// TIA Portal project "Giữa kì" (V15)

(* hardware
DEVICE "S7-1200 station_1"  S7-1200 Station
   slot 0: "Rack_0"  S7-1200 Rack  Rack  V1.0
   slot 1: "PLC_1"  CPU 1214C DC/DC/DC  6ES7 214-1AG40-0XB0  V4.2
*)

// ===== PLC "PLC_1"  CPU 1214C DC/DC/DC =====

VAR_GLOBAL   // PLC tag table "Default tag table"
   "enableSystem" AT %M0.0 : Bool;
   "iStart" AT %M0.1 : Bool;
   "iStop" AT %M0.2 : Bool;
   "oPump1" AT %Q0.0 : Bool;
   "oPump2" AT %Q0.1 : Bool;
   "mRespond" AT %M0.3 : Bool;
   "iSensorHigh1" AT %M0.4 : Bool;
   "iSensorLow1" AT %M0.5 : Bool;
   "Tag_1" AT %M100.0 : Bool;
   "Tag_2" AT %M100.1 : Bool;
   "mTank1" AT %M0.6 : Bool;
   "oPump3" AT %Q0.2 : Bool;
   "oValve1" AT %Q0.4 : Bool;
   "iSensorHigh3" AT %M1.1 : Bool;
   "iSensorLow3" AT %M1.2 : Bool;
   "iSensorHigh2" AT %M1.3 : Bool;
   "iSensorLow2" AT %M1.4 : Bool;
   "iSensorHigh4" AT %M1.5 : Bool;
   "iSensorLow4" AT %M1.6 : Bool;
   "mTank2" AT %M1.7 : Bool;
   "Tag_3" AT %M100.2 : Bool;
   "Tag_4" AT %M100.3 : Bool;
   "Tag_5" AT %M100.4 : Bool;
   "Tag_6" AT %M100.5 : Bool;
   "mTank3" AT %M2.0 : Bool;
   "mTank4" AT %M2.1 : Bool;
   "oValve2" AT %Q0.5 : Bool;
   "Tag_7" AT %M100.6 : Bool;
   "oPump4" AT %Q0.3 : Bool;
   "Tag_8" AT %M100.7 : Bool;
END_VAR

DATA_BLOCK "Data_block_1"   // DB3
{ S7_Optimized_Access := 'TRUE' }
VERSION : 0.1
   VAR
      RequiredSalinity : Real := 3.0;
      ActualSalinity : Real := 4.0;
   END_VAR
BEGIN
END_DATA_BLOCK

// folder: System blocks/Program resources

DATA_BLOCK "TimerPump1"   // DB1
{ S7_Optimized_Access := 'TRUE' }
AUTHOR : Simatic
FAMILY : IEC
NAME : IEC_TMR
VERSION : 1.0
// stored: InstanceOfName IEC_TIMER
"IEC_TIMER"
BEGIN
END_DATA_BLOCK

DATA_BLOCK "TimerPump2"   // DB2
{ S7_Optimized_Access := 'TRUE' }
AUTHOR : Simatic
FAMILY : IEC
NAME : IEC_TMR
VERSION : 1.0
// stored: InstanceOfName IEC_TIMER
"IEC_TIMER"
BEGIN
END_DATA_BLOCK

// folder: (top level)

ORGANIZATION_BLOCK "Main"   // OB1, LAD, ProgramCycle
TITLE = "Main Program Sweep (Cycle)"
{ S7_Optimized_Access := 'TRUE' }
VERSION : 0.1
   VAR_INPUT
      Initial_Call : Bool;   // Initial call of this OB
      Remanence : Bool;   // =True, if remanent data are available
   END_VAR
   VAR_TEMP   // added for the SCL form of the ladder/FBD networks
      _w1 : Bool;
      _w2 : Bool;
   END_VAR
BEGIN

REGION Network 1
   // Mở và tắt hệ thống
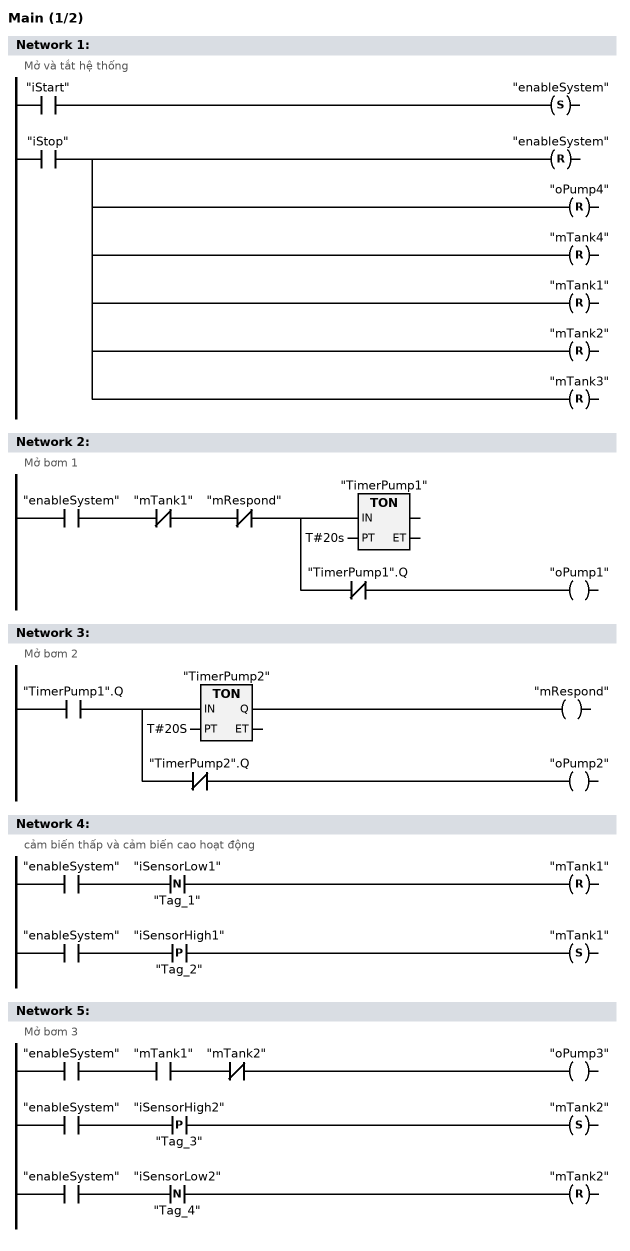
   RUNG wire#powerrail
      Contact( "iStart" )
      S_Coil( "enableSystem" )
   END_RUNG
   RUNG wire#powerrail
      Contact( "iStop" )
      wire#w1
      R_Coil( "enableSystem" )
   END_RUNG
   RUNG wire#w1
      R_Coil( "oPump4" )
   END_RUNG
   RUNG wire#w1
      R_Coil( "mTank4" )
   END_RUNG
   RUNG wire#w1
      R_Coil( "mTank1" )
   END_RUNG
   RUNG wire#w1
      R_Coil( "mTank2" )
   END_RUNG
   RUNG wire#w1
      R_Coil( "mTank3" )
   END_RUNG
   // the same network as SCL:
   IF "iStart" THEN "enableSystem" := TRUE; END_IF;
   IF "iStop" THEN
       "enableSystem" := FALSE;
       "oPump4" := FALSE;
       "mTank4" := FALSE;
       "mTank1" := FALSE;
       "mTank2" := FALSE;
       "mTank3" := FALSE;
   END_IF;
END_REGION

REGION Network 2
   // Mở bơm 1
   #_w1 := "enableSystem" AND NOT "mTank1" AND NOT "mRespond";
   "TimerPump1".TON(IN := #_w1, PT := T#20s);
   "oPump1" := #_w1 AND NOT "TimerPump1".Q;
END_REGION

REGION Network 3
   // Mở bơm 2
   "TimerPump2".TON(IN := "TimerPump1".Q, PT := T#20S);
   "mRespond" := "TimerPump2".Q;
   "oPump2" := "TimerPump1".Q AND NOT "TimerPump2".Q;
END_REGION

REGION Network 4
   // cảm biến thấp và cảm biến cao hoạt động
   RUNG wire#powerrail
      Contact( "enableSystem" )
      N_Contact(operand := "iSensorLow1", bit := "Tag_1")
      R_Coil( "mTank1" )
   END_RUNG
   RUNG wire#powerrail
      Contact( "enableSystem" )
      P_Contact(operand := "iSensorHigh1", bit := "Tag_2")
      S_Coil( "mTank1" )
   END_RUNG
   // the same network as SCL:
   #_w1 := "enableSystem" AND NOT "iSensorLow1" AND "Tag_1";   // falling edge of "iSensorLow1"
   "Tag_1" := "iSensorLow1";
   IF #_w1 THEN "mTank1" := FALSE; END_IF;
   #_w2 := "enableSystem" AND "iSensorHigh1" AND NOT "Tag_2";   // rising edge of "iSensorHigh1"
   "Tag_2" := "iSensorHigh1";
   IF #_w2 THEN "mTank1" := TRUE; END_IF;
END_REGION

REGION Network 5
   // Mở bơm 3
   RUNG wire#powerrail
      Contact( "enableSystem" )
      Contact( "mTank1" )
      I_Contact( "mTank2" )
      Coil( "oPump3" )
   END_RUNG
   RUNG wire#powerrail
      Contact( "enableSystem" )
      P_Contact(operand := "iSensorHigh2", bit := "Tag_3")
      S_Coil( "mTank2" )
   END_RUNG
   RUNG wire#powerrail
      Contact( "enableSystem" )
      N_Contact(operand := "iSensorLow2", bit := "Tag_4")
      R_Coil( "mTank2" )
   END_RUNG
   // the same network as SCL:
   "oPump3" := "enableSystem" AND "mTank1" AND NOT "mTank2";
   #_w1 := "enableSystem" AND "iSensorHigh2" AND NOT "Tag_3";   // rising edge of "iSensorHigh2"
   "Tag_3" := "iSensorHigh2";
   IF #_w1 THEN "mTank2" := TRUE; END_IF;
   #_w2 := "enableSystem" AND NOT "iSensorLow2" AND "Tag_4";   // falling edge of "iSensorLow2"
   "Tag_4" := "iSensorLow2";
   IF #_w2 THEN "mTank2" := FALSE; END_IF;
END_REGION

REGION Network 6
   // Mở van 1 cho nước xuống bể 3
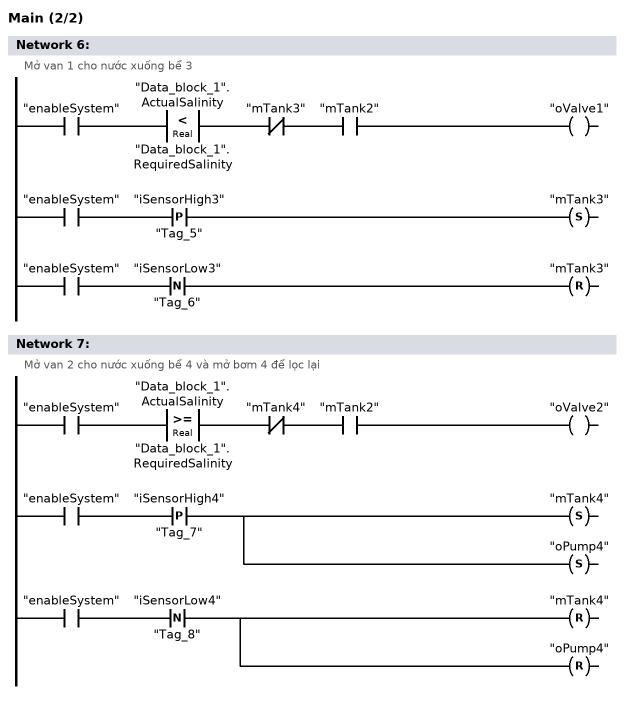
   RUNG wire#powerrail
      Contact( "enableSystem" )
      { S7_Templates := "SrcType := Real" } LT_Contact(in1 := "Data_block_1".ActualSalinity, in2 := "Data_block_1".RequiredSalinity)
      I_Contact( "mTank3" )
      Contact( "mTank2" )
      Coil( "oValve1" )
   END_RUNG
   RUNG wire#powerrail
      Contact( "enableSystem" )
      P_Contact(operand := "iSensorHigh3", bit := "Tag_5")
      S_Coil( "mTank3" )
   END_RUNG
   RUNG wire#powerrail
      Contact( "enableSystem" )
      N_Contact(operand := "iSensorLow3", bit := "Tag_6")
      R_Coil( "mTank3" )
   END_RUNG
   // the same network as SCL:
   "oValve1" := "enableSystem" AND ("Data_block_1".ActualSalinity < "Data_block_1".RequiredSalinity) AND NOT "mTank3" AND "mTank2";
   #_w1 := "enableSystem" AND "iSensorHigh3" AND NOT "Tag_5";   // rising edge of "iSensorHigh3"
   "Tag_5" := "iSensorHigh3";
   IF #_w1 THEN "mTank3" := TRUE; END_IF;
   #_w2 := "enableSystem" AND NOT "iSensorLow3" AND "Tag_6";   // falling edge of "iSensorLow3"
   "Tag_6" := "iSensorLow3";
   IF #_w2 THEN "mTank3" := FALSE; END_IF;
END_REGION

REGION Network 7
   // Mở van 2 cho nước xuống bể 4 và mở bơm 4 để lọc lại
   RUNG wire#powerrail
      Contact( "enableSystem" )
      { S7_Templates := "SrcType := Real" } GE_Contact(in1 := "Data_block_1".ActualSalinity, in2 := "Data_block_1".RequiredSalinity)
      I_Contact( "mTank4" )
      Contact( "mTank2" )
      Coil( "oValve2" )
   END_RUNG
   RUNG wire#powerrail
      Contact( "enableSystem" )
      P_Contact(operand := "iSensorHigh4", bit := "Tag_7")
      wire#w1
      S_Coil( "mTank4" )
   END_RUNG
   RUNG wire#w1
      S_Coil( "oPump4" )
   END_RUNG
   RUNG wire#powerrail
      Contact( "enableSystem" )
      N_Contact(operand := "iSensorLow4", bit := "Tag_8")
      wire#w2
      R_Coil( "mTank4" )
   END_RUNG
   RUNG wire#w2
      R_Coil( "oPump4" )
   END_RUNG
   // the same network as SCL:
   "oValve2" := "enableSystem" AND ("Data_block_1".ActualSalinity >= "Data_block_1".RequiredSalinity) AND NOT "mTank4" AND "mTank2";
   #_w1 := "enableSystem" AND "iSensorHigh4" AND NOT "Tag_7";   // rising edge of "iSensorHigh4"
   "Tag_7" := "iSensorHigh4";
   IF #_w1 THEN
       "mTank4" := TRUE;
       "oPump4" := TRUE;
   END_IF;
   #_w2 := "enableSystem" AND NOT "iSensorLow4" AND "Tag_8";   // falling edge of "iSensorLow4"
   "Tag_8" := "iSensorLow4";
   IF #_w2 THEN
       "mTank4" := FALSE;
       "oPump4" := FALSE;
   END_IF;
END_REGION
END_ORGANIZATION_BLOCK